% RSLogix 500 project PUMP_PROTECTION.RSS, saved by version 8.30.00.16 %
PROJECT "UNTITLED"    % processor: Bul.1763 MicroLogix 1100 Series B %

PROGRAM FILES
  LAD 2 "MAIN"  7 rungs
  LAD 3 "I/O"  11 rungs
  LAD 4 "CYCLE"  3 rungs
  LAD 5 "ALARMS"  5 rungs
  LAD 6 "CONTROL"  5 rungs

DATA FILES
  O0 OUTPUT  7 elements
  I1 INPUT  13 elements
  S2 STATUS  66 elements
  B3 BINARY  2 elements
  T4 TIMER  4 elements
  C5 COUNTER  1 elements
  R6 CONTROL  1 elements
  N7 INTEGER  5 elements
  F8 FLOAT  1 elements

LADDER 2 "MAIN"
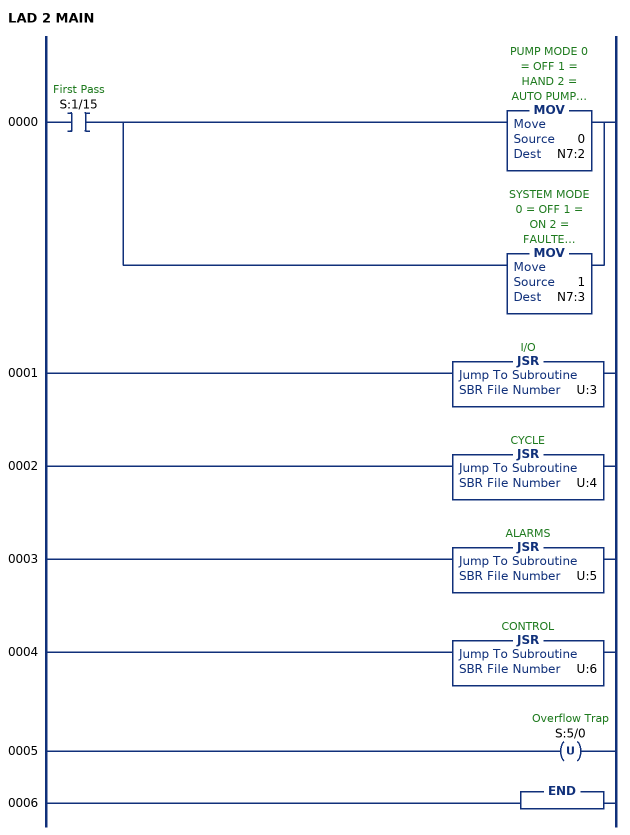
% Rung: 0 %
SOR XIC S:1/15 BST MOV 0 N7:2 NXB MOV 1 N7:3 BND EOR
%   S:1/15  "First Pass" %
%   N7:2  PUMP_MODE  "PUMP MODE 0 = OFF 1 = HAND 2 = AUTO" %
%   N7:3  SYSTEM_MODE  "SYSTEM MODE 0 = OFF 1 = ON 2 = FAULTED" %
% Rung: 1 %
SOR JSR U:3 EOR
%   U:3  "I/O" %
% Rung: 2 %
SOR JSR U:4 EOR
%   U:4  "CYCLE" %
% Rung: 3 %
SOR JSR U:5 EOR
%   U:5  "ALARMS" %
% Rung: 4 %
SOR JSR U:6 EOR
%   U:6  "CONTROL" %
% Rung: 5 %
SOR OTU S:5/0 EOR
%   S:5/0  "Overflow Trap" %
% Rung: 6 %
SOR END EOR

LADDER 3 "I/O"
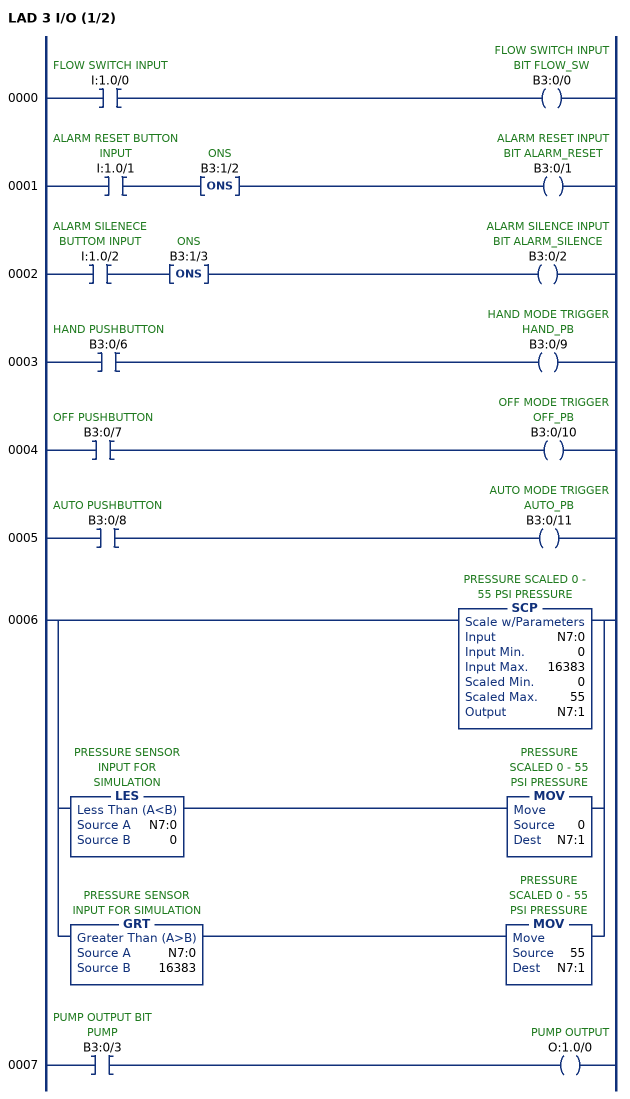
% Rung: 0 %
SOR XIC I:1.0/0 OTE B3:0/0 EOR
%   I:1.0/0  "FLOW SWITCH INPUT" %
%   B3:0/0  FLOW_SW  "FLOW SWITCH INPUT BIT" %
% Rung: 1 %
SOR XIC I:1.0/1 ONS B3:1/2 OTE B3:0/1 EOR
%   I:1.0/1  "ALARM RESET BUTTON INPUT" %
%   B3:1/2  "ONS" %
%   B3:0/1  ALARM_RESET  "ALARM RESET INPUT BIT" %
% Rung: 2 %
SOR XIC I:1.0/2 ONS B3:1/3 OTE B3:0/2 EOR
%   I:1.0/2  "ALARM SILENECE BUTTOM INPUT" %
%   B3:1/3  "ONS" %
%   B3:0/2  ALARM_SILENCE  "ALARM SILENCE INPUT BIT" %
% Rung: 3 %
SOR XIC B3:0/6 OTE B3:0/9 EOR
%   B3:0/6  "HAND PUSHBUTTON" %
%   B3:0/9  HAND_PB  "HAND MODE TRIGGER" %
% Rung: 4 %
SOR XIC B3:0/7 OTE B3:0/10 EOR
%   B3:0/7  "OFF PUSHBUTTON" %
%   B3:0/10  OFF_PB  "OFF MODE TRIGGER" %
% Rung: 5 %
SOR XIC B3:0/8 OTE B3:0/11 EOR
%   B3:0/8  "AUTO PUSHBUTTON" %
%   B3:0/11  AUTO_PB  "AUTO MODE TRIGGER" %
% Rung: 6 %
SOR BST SCP N7:0 0 16383 0 55 N7:1 NXB LES N7:0 0 MOV 0 N7:1 NXB GRT N7:0 16383 MOV 55 N7:1 BND EOR
%   N7:0  "PRESSURE SENSOR INPUT FOR SIMULATION" %
%   N7:1  PRESSURE  "PRESSURE SCALED 0 - 55 PSI" %
% Rung: 7 %
SOR XIC B3:0/3 OTE O:1.0/0 EOR
%   B3:0/3  PUMP  "PUMP OUTPUT BIT" %
%   O:1.0/0  "PUMP OUTPUT" %

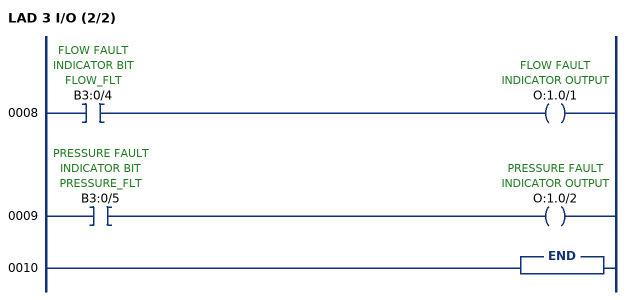
% Rung: 8 %
SOR XIC B3:0/4 OTE O:1.0/1 EOR
%   B3:0/4  FLOW_FLT  "FLOW FAULT INDICATOR BIT" %
%   O:1.0/1  "FLOW FAULT INDICATOR OUTPUT" %
% Rung: 9 %
SOR XIC B3:0/5 OTE O:1.0/2 EOR
%   B3:0/5  PRESSURE_FLT  "PRESSURE FAULT INDICATOR BIT" %
%   O:1.0/2  "PRESSURE FAULT INDICATOR OUTPUT" %
% Rung: 10 %
SOR END EOR

LADDER 4 "CYCLE"
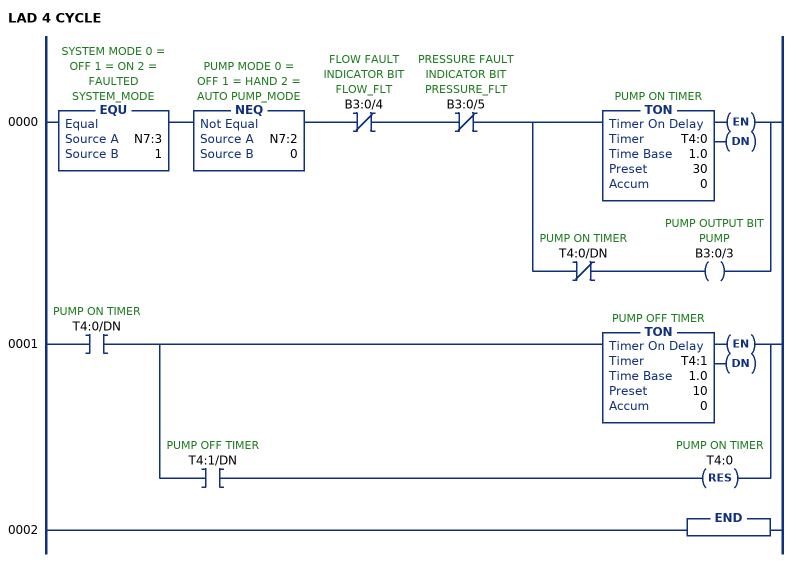
% Rung: 0 %
SOR EQU N7:3 1 NEQ N7:2 0 XIO B3:0/4 XIO B3:0/5 BST TON T4:0 1.0 30 0 NXB XIO T4:0/DN OTE B3:0/3 BND EOR
%   N7:3  SYSTEM_MODE  "SYSTEM MODE 0 = OFF 1 = ON 2 = FAULTED" %
%   N7:2  PUMP_MODE  "PUMP MODE 0 = OFF 1 = HAND 2 = AUTO" %
%   B3:0/4  FLOW_FLT  "FLOW FAULT INDICATOR BIT" %
%   B3:0/5  PRESSURE_FLT  "PRESSURE FAULT INDICATOR BIT" %
%   T4:0  "PUMP ON TIMER" %
%   B3:0/3  PUMP  "PUMP OUTPUT BIT" %
% Rung: 1 %
SOR XIC T4:0/DN BST TON T4:1 1.0 10 0 NXB XIC T4:1/DN RES T4:0 BND EOR
%   T4:0  "PUMP ON TIMER" %
%   T4:1  "PUMP OFF TIMER" %
% Rung: 2 %
SOR END EOR

LADDER 5 "ALARMS"
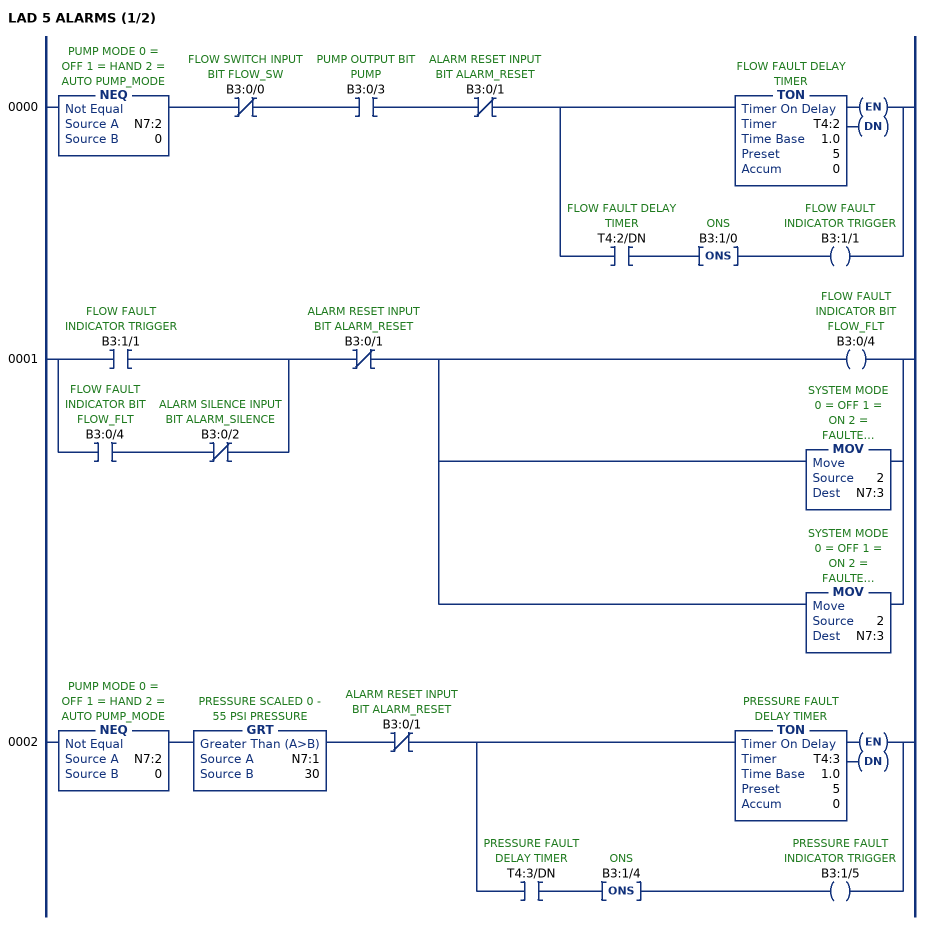
% Rung: 0 %
SOR NEQ N7:2 0 XIO B3:0/0 XIC B3:0/3 XIO B3:0/1 BST TON T4:2 1.0 5 0 NXB XIC T4:2/DN ONS B3:1/0 OTE B3:1/1 BND EOR
%   N7:2  PUMP_MODE  "PUMP MODE 0 = OFF 1 = HAND 2 = AUTO" %
%   B3:0/0  FLOW_SW  "FLOW SWITCH INPUT BIT" %
%   B3:0/3  PUMP  "PUMP OUTPUT BIT" %
%   B3:0/1  ALARM_RESET  "ALARM RESET INPUT BIT" %
%   T4:2  "FLOW FAULT DELAY TIMER" %
%   B3:1/0  "ONS" %
%   B3:1/1  "FLOW FAULT INDICATOR TRIGGER" %
% Rung: 1 %
SOR BST XIC B3:1/1 NXB XIC B3:0/4 XIO B3:0/2 BND XIO B3:0/1 BST OTE B3:0/4 NXB MOV 2 N7:3 NXB MOV 2 N7:3 BND EOR
%   B3:1/1  "FLOW FAULT INDICATOR TRIGGER" %
%   B3:0/4  FLOW_FLT  "FLOW FAULT INDICATOR BIT" %
%   B3:0/2  ALARM_SILENCE  "ALARM SILENCE INPUT BIT" %
%   B3:0/1  ALARM_RESET  "ALARM RESET INPUT BIT" %
%   N7:3  SYSTEM_MODE  "SYSTEM MODE 0 = OFF 1 = ON 2 = FAULTED" %
% Rung: 2 %
SOR NEQ N7:2 0 GRT N7:1 30 XIO B3:0/1 BST TON T4:3 1.0 5 0 NXB XIC T4:3/DN ONS B3:1/4 OTE B3:1/5 BND EOR
%   N7:2  PUMP_MODE  "PUMP MODE 0 = OFF 1 = HAND 2 = AUTO" %
%   N7:1  PRESSURE  "PRESSURE SCALED 0 - 55 PSI" %
%   B3:0/1  ALARM_RESET  "ALARM RESET INPUT BIT" %
%   T4:3  "PRESSURE FAULT DELAY TIMER" %
%   B3:1/4  "ONS" %
%   B3:1/5  "PRESSURE FAULT INDICATOR TRIGGER" %

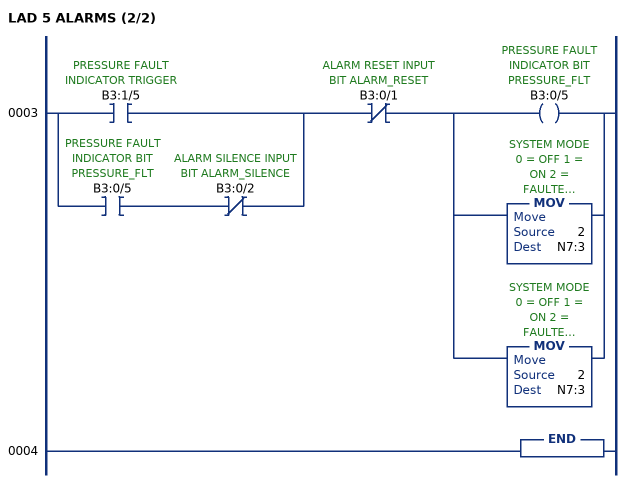
% Rung: 3 %
SOR BST XIC B3:1/5 NXB XIC B3:0/5 XIO B3:0/2 BND XIO B3:0/1 BST OTE B3:0/5 NXB MOV 2 N7:3 NXB MOV 2 N7:3 BND EOR
%   B3:1/5  "PRESSURE FAULT INDICATOR TRIGGER" %
%   B3:0/5  PRESSURE_FLT  "PRESSURE FAULT INDICATOR BIT" %
%   B3:0/2  ALARM_SILENCE  "ALARM SILENCE INPUT BIT" %
%   B3:0/1  ALARM_RESET  "ALARM RESET INPUT BIT" %
%   N7:3  SYSTEM_MODE  "SYSTEM MODE 0 = OFF 1 = ON 2 = FAULTED" %
% Rung: 4 %
SOR END EOR

LADDER 6 "CONTROL"
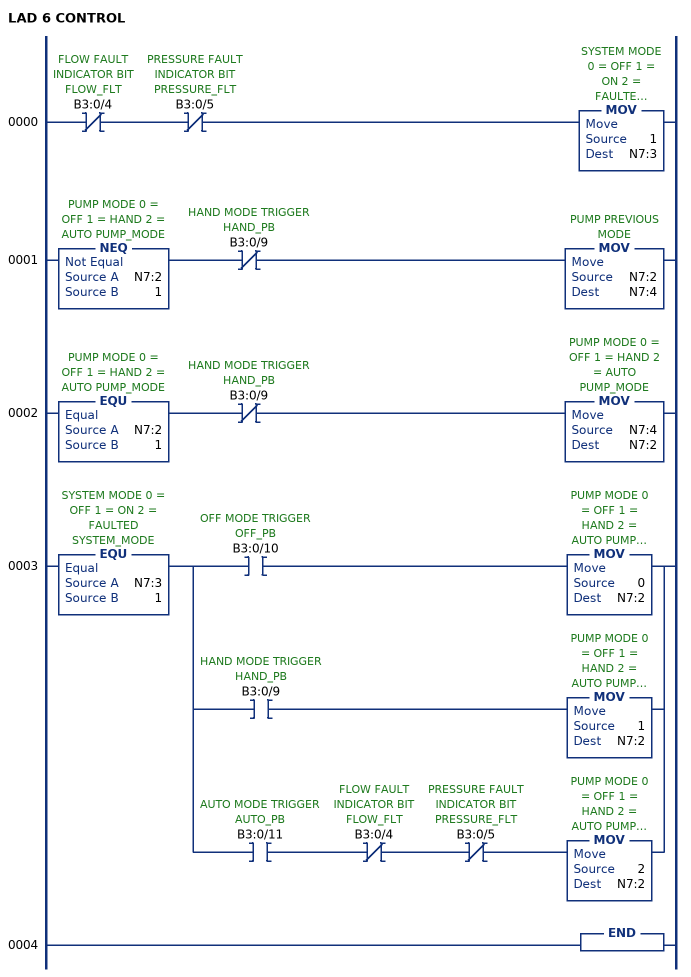
% Rung: 0 %
SOR XIO B3:0/4 XIO B3:0/5 MOV 1 N7:3 EOR
%   B3:0/4  FLOW_FLT  "FLOW FAULT INDICATOR BIT" %
%   B3:0/5  PRESSURE_FLT  "PRESSURE FAULT INDICATOR BIT" %
%   N7:3  SYSTEM_MODE  "SYSTEM MODE 0 = OFF 1 = ON 2 = FAULTED" %
% Rung: 1 %
SOR NEQ N7:2 1 XIO B3:0/9 MOV N7:2 N7:4 EOR
%   N7:2  PUMP_MODE  "PUMP MODE 0 = OFF 1 = HAND 2 = AUTO" %
%   B3:0/9  HAND_PB  "HAND MODE TRIGGER" %
%   N7:4  "PUMP PREVIOUS MODE" %
% Rung: 2 %
SOR EQU N7:2 1 XIO B3:0/9 MOV N7:4 N7:2 EOR
%   N7:2  PUMP_MODE  "PUMP MODE 0 = OFF 1 = HAND 2 = AUTO" %
%   B3:0/9  HAND_PB  "HAND MODE TRIGGER" %
%   N7:4  "PUMP PREVIOUS MODE" %
% Rung: 3 %
SOR EQU N7:3 1 BST XIC B3:0/10 MOV 0 N7:2 NXB XIC B3:0/9 MOV 1 N7:2 NXB XIC B3:0/11 XIO B3:0/4 XIO B3:0/5 MOV 2 N7:2 BND EOR
%   N7:3  SYSTEM_MODE  "SYSTEM MODE 0 = OFF 1 = ON 2 = FAULTED" %
%   B3:0/10  OFF_PB  "OFF MODE TRIGGER" %
%   N7:2  PUMP_MODE  "PUMP MODE 0 = OFF 1 = HAND 2 = AUTO" %
%   B3:0/9  HAND_PB  "HAND MODE TRIGGER" %
%   B3:0/11  AUTO_PB  "AUTO MODE TRIGGER" %
%   B3:0/4  FLOW_FLT  "FLOW FAULT INDICATOR BIT" %
%   B3:0/5  PRESSURE_FLT  "PRESSURE FAULT INDICATOR BIT" %
% Rung: 4 %
SOR END EOR

OTHER DOCUMENTED ADDRESSES
  B3:1/6  "ONS"

DATA TABLE (non-zero values as saved)
DATA T4
% .PRE .ACC %
% T4:0 % 30 0
% T4:1 % 10 0
% T4:2 % 5 0
% T4:3 % 5 0
DATA N7
% N7:0 % 8192 0 0 0 0
